(*
SPDX-FileCopyrightText: © 2026 Oleksandr Tiutyk <trofimich@gmail.com>
SPDX-License-Identifier: MIT
License: https://opensource.org/license/mit
*)

FUNCTION_BLOCK ExceptionTest EXTENDS TcUnit.FB_TestSuite
VAR
	{attribute 'hide'} 
	_ClassName : STRING := __POUNAME();	
END_VAR

SimpleException();
StandardExceptions();
AggregateException();
RethrowSavedFrameworkException();
RethrowSystemExceptionAfterFramework();
TimestampFormatting();
SystemExceptionClone();
AggregateCloneLifetime();
ArgumentTypeCloneIdentity();

METHOD AggregateCloneLifetime
VAR
	source : TOF_Core.StandardException;
	aggregate : TOF_Core.AggregateException;
	dynamicInner : TOF_Core.IException;
	clonedObject : TOF_Core.IObject;
	clonedAggregate : TOF_Core.IAggregateException;
	firstInner : TOF_Core.IException;
	storedDynamicInner : TOF_Core.IException;
	clonedFirstInner : TOF_Core.IException;
	clonedSecondInner : TOF_Core.IException;
	caughtCode : __SYSTEM.ExceptionCode;
	caught : BOOL;
	queried : BOOL;
END_VAR
VAR_INST
	testFinished : BOOL;
END_VAR
IF testFinished THEN 
	RETURN; 
END_IF

TEST(__POUNAME());

__TRY
	source.Throw(NamespaceName, ClassName, __POUNAME(), __POSITION(), "Original inner");
__CATCH(caughtCode)
	caught := TRUE;
	dynamicInner := TOF_Core.ExceptionManager.GetLastException(caughtCode, NamespaceName, __POUNAME(), __POSITION());
__ENDTRY

AssertEquals_BOOL(TRUE, caught, 'Expected a dynamic exception from static Throw');

IF caught THEN
	aggregate.AddInnerException(source);
	aggregate.AddInnerException(dynamicInner);
	source.Clear();
	firstInner := aggregate.GetInnerException(0);
	AssertEquals_BOOL(TRUE, firstInner <> 0, 'Static inner must be cloned');
	
	IF firstInner <> 0 THEN
		AssertEquals_WSTRING("Original inner", firstInner.GetMessage(), 'Clearing static source must not clear the stored clone');
	END_IF
	
	storedDynamicInner := aggregate.GetInnerException(1);
	AssertEquals_BOOL(TRUE, storedDynamicInner = dynamicInner, 'Dynamic inner must retain identity');

	clonedObject := aggregate.Clone();
	queried := __QUERYINTERFACE(clonedObject, clonedAggregate);
	AssertEquals_BOOL(TRUE, queried, 'Aggregate clone must implement IAggregateException');

	aggregate.Clear();
	aggregate.Clear();

	AssertEquals_UINT(0, aggregate.InnerExceptionCount, 'Repeated Clear must leave an empty aggregate');
	IF queried THEN
		AssertEquals_UINT(2, clonedAggregate.InnerExceptionCount, 'Clearing source must preserve the clone array');

		clonedFirstInner := clonedAggregate.GetInnerException(0);
		clonedSecondInner := clonedAggregate.GetInnerException(1);

		AssertEquals_BOOL(TRUE, clonedFirstInner = firstInner AND_THEN clonedSecondInner = dynamicInner, 'Aggregate clone must borrow the same dynamic inners');
	END_IF
END_IF

// All dynamic exception instances are released by the manager at the cycle boundary.
testFinished := TRUE;
TEST_FINISHED();
END_METHOD

METHOD AggregateException
VAR
	caught : BOOL;
	exception1Message : WSTRING := "Simple exception 1 thrown";
	exception2Message : WSTRING := "Simple exception 2 thrown";
	exception3Message : WSTRING := "Simple exception 3 thrown";
	
	errorMessage : TOF_Core.ERROR_MESSAGE;
	
	standardException1 : TOF_Core.StandardException;
	standardException2 : TOF_Core.StandardException;
	standardException3 : TOF_Core.StandardException;

	exceptionCode : __SYSTEM.ExceptionCode;
	caughtException : TOF_Core.IException;
	
	aggregateException : TOF_Core.AggregateException;
END_VAR
VAR_INST
	testFinished : BOOL;
END_VAR
IF testFinished THEN 
	RETURN; 
END_IF 

TEST(__POUNAME());

caught := FALSE;
__TRY
	standardException1.Throw(NamespaceName, ClassName, __POUNAME(), __POSITION(), exception1Message, 0, 0);
__CATCH(exceptionCode)
	caught := TRUE;
	caughtException := TOF_Core.ExceptionManager.GetLastException(exceptionCode, NamespaceName, __POUNAME(), __POSITION());
	aggregateException.AddInnerException(caughtException);
__ENDTRY
AssertEquals_BOOL(TRUE, caught, 'Expected exception was not raised');

caught := FALSE;
__TRY
	standardException2.Throw(NamespaceName, ClassName, __POUNAME(), __POSITION(), exception2Message, 0, 0);
__CATCH(exceptionCode)
	caught := TRUE;
	caughtException := TOF_Core.ExceptionManager.GetLastException(exceptionCode, NamespaceName, __POUNAME(), __POSITION());
	aggregateException.AddInnerException(caughtException);
__ENDTRY
AssertEquals_BOOL(TRUE, caught, 'Expected exception was not raised');

caught := FALSE;
__TRY
	standardException3.Throw(NamespaceName, ClassName, __POUNAME(), __POSITION(), exception3Message, 0, 0);
__CATCH(exceptionCode)
	caught := TRUE;
	caughtException := TOF_Core.ExceptionManager.GetLastException(exceptionCode, NamespaceName, __POUNAME(), __POSITION());
	aggregateException.AddInnerException(caughtException);
__ENDTRY
AssertEquals_BOOL(TRUE, caught, 'Expected exception was not raised');

// for breakpoint
errorMessage := errorMessage;

caught := FALSE;
__TRY
	aggregateException.Throw(NamespaceName, ClassName, __POUNAME(), __POSITION());
__CATCH(exceptionCode)
	caught := TRUE;
	caughtException := TOF_Core.ExceptionManager.GetLastException(exceptionCode, NamespaceName, __POUNAME(), __POSITION());
	
	errorMessage := caughtException.GetMessage();
	
	AssertEquals_INT(1,	Tc2_Standard.WFIND(errorMessage, "3"), 'Wrong aggregate exception message caught');	
__ENDTRY
AssertEquals_BOOL(TRUE, caught, 'Expected exception was not raised');

testFinished := TRUE; 
TEST_FINISHED();
END_METHOD

METHOD ArgumentTypeCloneIdentity
VAR
	source : TOF_Core.ArgumentTypeNotSupportedException;
	clonedObject : TOF_Core.IObject;
	typedClone : TOF_Core.IArgumentTypeNotSupportedException;
END_VAR
VAR_INST
	testFinished : BOOL;
END_VAR
IF testFinished THEN 
	RETURN; 
END_IF

TEST(__POUNAME());

clonedObject := source.Clone();
AssertEquals_BOOL(TRUE, __QUERYINTERFACE(clonedObject, typedClone), 'Clone must preserve IArgumentTypeNotSupportedException');

// The dynamic clone is owned by DynamicMemoryManager.
testFinished := TRUE;
TEST_FINISHED();
END_METHOD

{attribute 'monitoring' := 'call'}
PROPERTY ClassName : REFERENCE TO STRING
GET
ClassName REF= _ClassName;
END_GET
END_PROPERTY

{attribute 'monitoring' := 'call'}
PROPERTY NamespaceName : REFERENCE TO STRING
GET
NamespaceName REF= CurrentNamespace.Name;
END_GET
END_PROPERTY

METHOD RethrowSavedFrameworkException
VAR
	original : TOF_Core.StandardException;
	nested : TOF_Core.StandardException;
	saved : TOF_Core.IException;
	received : TOF_Core.IException;
	caughtCode : __SYSTEM.ExceptionCode;
	outerCode : __SYSTEM.ExceptionCode;
	caught : BOOL;
END_VAR
VAR_INST
	testFinished : BOOL;
END_VAR
IF testFinished THEN 
	RETURN; 
END_IF

TEST(__POUNAME());

__TRY
	__TRY
		original.Throw(NamespaceName, ClassName, __POUNAME(), __POSITION(), "Original");
	__CATCH(caughtCode)
		saved := TOF_Core.ExceptionManager.GetLastException(caughtCode, NamespaceName, __POUNAME(), __POSITION());

		__TRY
			nested.Throw(NamespaceName, ClassName, __POUNAME(), __POSITION(), "Nested");
		__CATCH
		__ENDTRY

		TOF_Core.ExceptionManager.ReThrowLastException(caughtCode, saved);
	__ENDTRY
__CATCH(outerCode)
	caught := TRUE;
	received := TOF_Core.ExceptionManager.GetLastException(outerCode, NamespaceName, __POUNAME(), __POSITION());
__ENDTRY

AssertEquals_BOOL(TRUE, caught, 'Expected rethrown framework exception');
AssertEquals_BOOL(TRUE, saved <> 0 AND_THEN received = saved, 'Nested catch must not replace the saved payload');

testFinished := TRUE;
TEST_FINISHED();
END_METHOD

(*!
<summary>Checks SystemException propagation after a previous framework error, including nested handlers.</summary>
<description>
Supplies a known native code to the adapter without using F_RaiseException to generate the initial error.
This tests wrapper propagation; it does not verify delivery of the initial native code by TwinCAT.
</description>
*)
METHOD RethrowSystemExceptionAfterFramework
VAR
	previous : TOF_Core.StandardException;
	outerCode : __SYSTEM.ExceptionCode;
	original : TOF_Core.IException;
	received : TOF_Core.IException;
	repeated : TOF_Core.IException;
	otherSystem : TOF_Core.IException;
	expectedMessage : TOF_Core.ERROR_MESSAGE;
	savedLocalTime : LDATE_AND_TIME;
	savedUtcTime : LDATE_AND_TIME;
	caught : BOOL;
END_VAR
VAR_INST
	testFinished : BOOL;
END_VAR
IF testFinished THEN 
	RETURN; 
END_IF

TEST(__POUNAME());

__TRY
	previous.Throw(NamespaceName, ClassName, __POUNAME(), __POSITION(), "Previous");
__CATCH
__ENDTRY

// Model an already received native code; the runtime's initial raise bug is a separate limitation.
original := TOF_Core.ExceptionManager.GetLastException(__SYSTEM.ExceptionCode.RTSEXCPT_ARRAYBOUNDS, NamespaceName, 'OriginalCatch', 'OriginalPosition');
expectedMessage := original.GetMessage();
savedLocalTime := original.LocalTimestamp;
savedUtcTime := original.UtcTimestamp;

caught := FALSE;
__TRY
	TOF_Core.ExceptionManager.ReThrowLastException(__SYSTEM.ExceptionCode.RTSEXCPT_ARRAYBOUNDS, original);
__CATCH(outerCode)
	caught := TRUE;
	received := TOF_Core.ExceptionManager.GetLastException(outerCode, NamespaceName, 'OuterCatch', 'OuterPosition');
__ENDTRY

AssertEquals_BOOL(TRUE, caught, 'Expected propagated system wrapper');
AssertEquals_BOOL(TRUE, received <> 0, 'System wrapper must be available in the next catch');

IF received <> 0 THEN
	AssertEquals_BOOL(TRUE, received.IsDynamicInstance, 'Static system wrapper must be cloned for propagation');
	AssertEquals_BOOL(TRUE, received <> original, 'Propagated wrapper must be independent of shared storage');
	AssertEquals_WSTRING(expectedMessage, received.GetMessage(), 'Wrapper must retain native error and original catch point');
	AssertEquals_BOOL(TRUE, received.LocalTimestamp = savedLocalTime AND_THEN received.UtcTimestamp = savedUtcTime, 'Wrapper must retain original timestamps');

	otherSystem := TOF_Core.ExceptionManager.GetLastException(__SYSTEM.ExceptionCode.RTSEXCPT_ACCESS_VIOLATION, NamespaceName, 'OtherCatch', 'OtherPosition');
	AssertEquals_WSTRING(expectedMessage, received.GetMessage(), 'Another system catch must not overwrite the propagated wrapper');

	// Replace the manager payload before propagating the saved dynamic wrapper again.
	__TRY
		previous.Throw(NamespaceName, ClassName, __POUNAME(), __POSITION(), "Nested");
	__CATCH
	__ENDTRY
	
	caught := FALSE;
	
	__TRY
		TOF_Core.ExceptionManager.ReThrowLastException(__SYSTEM.ExceptionCode.RTSEXCPT_ARRAYBOUNDS, received);
	__CATCH(outerCode)
		caught := TRUE;
		repeated := TOF_Core.ExceptionManager.GetLastException(outerCode, NamespaceName, 'NextCatch', 'NextPosition');
	__ENDTRY
	
	AssertEquals_BOOL(TRUE, caught, 'Expected saved system wrapper to be propagated again');
	AssertEquals_BOOL(TRUE, repeated = received, 'Repeated propagation must retain the saved dynamic wrapper identity');
END_IF

// Callers without a saved payload supply the catch code and location directly.
caught := FALSE;
repeated := 0;

__TRY
	TOF_Core.ExceptionManager.ReThrowLastException(exceptionCode := __SYSTEM.ExceptionCode.RTSEXCPT_ARRAYBOUNDS, catchPointNamespaceName := NamespaceName, catchPointPOUName := 'OriginalCatch', catchPointPosition := 'OriginalPosition');
__CATCH(outerCode)
	caught := TRUE;
	repeated := TOF_Core.ExceptionManager.GetLastException(outerCode, NamespaceName, 'OuterCatch', 'OuterPosition');
__ENDTRY

AssertEquals_BOOL(TRUE, caught, 'Expected native code to be wrapped without a supplied payload');
AssertEquals_BOOL(TRUE, repeated <> 0, 'Expected a wrapper for the supplied native code');

IF repeated <> 0 THEN
	AssertEquals_WSTRING(expectedMessage, repeated.GetMessage(), 'Code-only propagation must preserve native error and catch point');
END_IF

// Dynamic wrappers belong to DynamicMemoryManager until cycle cleanup.
testFinished := TRUE;
TEST_FINISHED();
END_METHOD

//!<param name="exceptionCode">filled by __CATCH statement</param>

//!<param name="exception">exception object returned by ExceptionManager</param>

//!<param name="notImplementedException">to filter specific exception type</param>

//!<param name="exceptionMessage">exception message</param>

METHOD SimpleException
VAR
	caught : BOOL;
	exceptionCode : __SYSTEM.ExceptionCode; 
	
	exception : TOF_Core.IException; 
	
	notImplementedException : TOF_Core.INotImplementedException; 
	
	exceptionMessage : WSTRING(255); 
END_VAR
VAR_INST
	testFinished : BOOL;
END_VAR
IF testFinished THEN 
	RETURN; 
END_IF 

TEST(__POUNAME());

caught := FALSE;

__TRY	
	throwNotImplementedException(); // your logic
__CATCH(exceptionCode)
	caught := TRUE;
	exception := TOF_Core.ExceptionManager.GetLastException(exceptionCode, NamespaceName, __POUNAME(), __POSITION()); // get exception object

	IF __QUERYINTERFACE(exception, notImplementedException) THEN // check if exception is of NotImplemented class
		exceptionMessage := notImplementedException.GetMessage(); // Get exception message	

		AssertEquals_WSTRING("Program organization unit 'TOF_Tests.ExceptionTest.throwNotImplementedException()' is not implemented", exceptionMessage, 'Wrong NotImplementedException message');
	ELSE
		AssertEquals_BOOL(TRUE, FALSE, 'Wrong exception class'); // handle all other exceptions
	END_IF
__ENDTRY

AssertEquals_BOOL(TRUE, caught, 'Expected exception was not raised');

testFinished := TRUE; 
TEST_FINISHED();
END_METHOD

METHOD StandardExceptions
VAR
	caught : BOOL;
	exception1Message : WSTRING := "Simple exception 1";
	exception2Message : WSTRING := "Simple exception 2";
	exception3Message : WSTRING := "Simple exception 3";
	
	expectedErrorMessage : WSTRING(255);
	recievedErrorMessage : WSTRING(255);
	
	standardException1 : TOF_Core.StandardException;
	standardException2 : TOF_Core.StandardException;
	standardException3 : TOF_Core.StandardException;
	
	caughtException : TOF_Core.IException;
	
	exceptionCode : __SYSTEM.ExceptionCode;
END_VAR
VAR_INST
	testFinished : BOOL;
END_VAR
IF testFinished THEN 
	RETURN; 
END_IF 

TEST(__POUNAME());

caught := FALSE;

__TRY
	standardException1.Throw(NamespaceName, ClassName, __POUNAME(), __POSITION(), exception1Message, 0, 0);
__CATCH(exceptionCode)
	caught := TRUE;
	caughtException := TOF_Core.ExceptionManager.GetLastException(exceptionCode, NamespaceName, __POUNAME(), __POSITION());
	
	expectedErrorMessage := exception2Message;
	recievedErrorMessage := caughtException.GetMessage();
	
	AssertEquals_WSTRING(
		exception1Message, 
		recievedErrorMessage, 
		'Wrong exception1 message caught');	
__ENDTRY

AssertEquals_BOOL(TRUE, caught, 'Expected exception was not raised');

caught := FALSE;
__TRY
	standardException2.Throw(NamespaceName, ClassName, __POUNAME(), __POSITION(), exception2Message, 0, caughtException);
__CATCH(exceptionCode)
	caught := TRUE;
	caughtException := TOF_Core.ExceptionManager.GetLastException(exceptionCode, NamespaceName, __POUNAME(), __POSITION());
	
	expectedErrorMessage := TOF_Core.WideStrings.Concat255(exception2Message, " -> ", exception1Message);
	recievedErrorMessage := caughtException.GetMessage();
	
	AssertEquals_WSTRING(
		expectedErrorMessage, 
		recievedErrorMessage, 
		'Wrong exception2 message caught');	
__ENDTRY

AssertEquals_BOOL(TRUE, caught, 'Expected exception was not raised');

caught := FALSE;
__TRY
	standardException3.Throw(NamespaceName, ClassName, __POUNAME(), __POSITION(), exception3Message, 0, caughtException);
__CATCH(exceptionCode)
	caught := TRUE;
	caughtException := TOF_Core.ExceptionManager.GetLastException(exceptionCode, NamespaceName, __POUNAME(), __POSITION());
	
	expectedErrorMessage := TOF_Core.WideStrings.Concat255(exception3Message, " -> ", exception2Message, " -> ", exception1Message);
	recievedErrorMessage := caughtException.GetMessage();
	
	AssertEquals_WSTRING(
		expectedErrorMessage, 
		recievedErrorMessage, 
		'Wrong exception3 message caught');	
__ENDTRY

AssertEquals_BOOL(TRUE, caught, 'Expected exception was not raised');

testFinished := TRUE; 
TEST_FINISHED();
END_METHOD

METHOD SystemExceptionClone
VAR
	original : TOF_Core.IException;
	clonedObject : TOF_Core.IObject;
	clonedException : TOF_Core.IException;
	queried : BOOL;
	message : TOF_Core.ERROR_MESSAGE;
	savedLocalTime : LDATE_AND_TIME;
	savedUtcTime : LDATE_AND_TIME;
END_VAR
VAR_INST
	testFinished : BOOL;
END_VAR
IF testFinished THEN 
	RETURN; 
END_IF

TEST(__POUNAME());

original := TOF_Core.ExceptionManager.GetLastException(__SYSTEM.ExceptionCode.RTSEXCPT_OUT_OF_MEMORY, 'CloneTest', 'OriginalCatch', 'P1');
message := original.GetMessage();
savedLocalTime := original.LocalTimestamp;
savedUtcTime := original.UtcTimestamp;

clonedObject := original.Clone();

queried := __QUERYINTERFACE(clonedObject, clonedException);
AssertEquals_BOOL(TRUE, queried, 'System clone must implement IException');

IF queried THEN
	AssertEquals_BOOL(TRUE, clonedException.IsDynamicInstance, 'System clone must be dynamic');
	// Reconfigure the shared system instance; the clone must retain the original catch point.
	original := TOF_Core.ExceptionManager.GetLastException(__SYSTEM.ExceptionCode.RTSEXCPT_NOEXCEPTION, 'Changed', 'Changed', 'P2');
	AssertEquals_WSTRING(message, clonedException.GetMessage(), 'System clone must preserve code and catch point');
	AssertEquals_BOOL(TRUE, clonedException.LocalTimestamp = savedLocalTime AND_THEN clonedException.UtcTimestamp = savedUtcTime, 'System clone must preserve occurrence timestamps');
END_IF

// The clone belongs to DynamicMemoryManager. Do not release it manually.
testFinished := TRUE;
TEST_FINISHED();
END_METHOD

METHOD PRIVATE throwNotImplementedException
VAR
	notImplementedException : TOF_Core.NotImplementedException;
END_VAR
notImplementedException.Throw(NamespaceName, ClassName, __POUNAME(), __POSITION());
END_METHOD

METHOD TimestampFormatting
VAR
	message : TOF_Core.ERROR_MESSAGE;
END_VAR
VAR_INST
	probe : ExceptionTimestampProbe;
	testFinished : BOOL;
END_VAR
VAR CONSTANT
	localTime : LDATE_AND_TIME := LDT#2026-10-06-15:04:05;
	utcTime : LDATE_AND_TIME := LDT#2026-10-06-12:04:05;
END_VAR
IF testFinished THEN 
	RETURN; 
END_IF

TEST(__POUNAME());

message := probe.FormatTimestamp(TOF_Core.TIMESTAMP_DISPLAY_MODE.HIDDEN, localTime, utcTime);
AssertEquals_WSTRING("", message, 'Hidden timestamp must produce no text');

message := probe.FormatTimestamp(TOF_Core.TIMESTAMP_DISPLAY_MODE.LOCAL, localTime, utcTime);
AssertEquals_BOOL(TRUE, Tc2_Standard.WFIND(message, "15:04:05") > 0, 'Local mode must use local time');
AssertEquals_BOOL(TRUE, Tc2_Standard.WFIND(message, "UTC") = 0, 'Local mode must not have a UTC suffix');

message := probe.FormatTimestamp(TOF_Core.TIMESTAMP_DISPLAY_MODE.UTC, localTime, utcTime);
AssertEquals_BOOL(TRUE, Tc2_Standard.WFIND(message, "12:04:05") > 0, 'UTC mode must use UTC time');
AssertEquals_WSTRING("UTC", Tc2_Standard.WRIGHT(message, 3), 'UTC suffix must survive timestamp truncation');

testFinished := TRUE;
TEST_FINISHED();
END_METHOD

END_FUNCTION_BLOCK

(* stored: Version 1.1.0.1, ProductVersion 3.1.4026.21
   POU ExceptionTest: Id {26e3c0f6-79be-0fd8-2416-047495069edc}, SpecialFunc None
   Method AggregateCloneLifetime: Id {b99d5e1b-9b7e-4c6c-ae5b-f36a74aebdd2}
   Method AggregateException: Id {a0a36685-039a-455b-9e90-8d283dc9d749}
   Method ArgumentTypeCloneIdentity: Id {35cd05cb-95a0-46b6-a37e-a04b522270db}
   Property ClassName: Id {111a4a8b-8aa4-412d-9e90-ebb90980416c}
   Get Get: Id {96410920-4b2e-41a3-b06d-e24debc1540a}
   Property NamespaceName: Id {b777c1c9-58c7-49aa-9113-7972a528cd45}
   Get Get: Id {a01d58c4-3aa8-4890-9401-b209dd4a14a3}
   Method RethrowSavedFrameworkException: Id {1392d859-48c4-418d-bce1-a5d8e9d1aa50}
   Method RethrowSystemExceptionAfterFramework: Id {ed6d4170-4d0a-448f-95f1-92495e20ca2e}
   Method SimpleException: Id {68b793dc-aa3d-48fc-b926-e787c555c9b4}
   Method StandardExceptions: Id {c3d65c3a-6585-4f11-ab6e-5902e1fc565c}
   Method SystemExceptionClone: Id {3200f00a-26ae-4015-a0c7-0b96c15b71ce}
   Method throwNotImplementedException: Id {812cab99-b998-4b88-8bd1-6a55f32844fc}
   Method TimestampFormatting: Id {c65b5cb7-89c0-49a5-bd2f-0f0ddba4cfdd} *)
